FUNCTION_BLOCK SM_LineRegulator EXTENDS StateMachine
VAR_INPUT
	 sSubscription1 : STRING(8);
	 sSubscription2 : STRING(8);
	 sSubscription3 : STRING(8);
END_VAR
VAR_OUTPUT
END_VAR
VAR
	fbTurntable : Turntable;

	aRollerConveyors : ARRAY[1..3] OF RollerConveyor;
	fbRollerConveyorExit : RollerConveyor;
	fbReadyStepWorker : FB_StepWorker;
	fbBusyStepWorker : FB_StepWorker;
	fbInitStepWorker : FB_StepWorker;
	
	messageIndex : UINT;
	stMqttPayload : ST_MqttPayload;
	aSubscriptions : ARRAY[1..3] OF STRING(8);
	uiSubscriptionsCycler : UINT := 1;
END_VAR

SUPER^();
fbTurntable();
aRollerConveyors[1]();
aRollerConveyors[3]();

METHOD PROTECTED   Busy : BOOL
VAR_INPUT
END_VAR
fbBusyStepWorker();
CASE fbBusyStepWorker.uiStep OF

	0:
	
		aRollerConveyors[uiSubscriptionsCycler].On();
		CASE uiSubscriptionsCycler OF
		
			1:
				fbTurntable.RollPlus();
				fbTurntable.Turn();
			
			2:
				fbTurntable.RollPlus();
			
			3:
				fbTurntable.RollMinus();
				fbTurntable.Turn();
		END_CASE
		
		fbBusyStepWorker
			.mAddCondition(itfStepCondition := fbTurntable.fbBackLimit.getSignal)
			.mAddCondition(itfStepCondition := fbTurntable.fbFrontLimit.getSignal)
			.mNextStep(10);
			
	10:
	
		aRollerConveyors[uiSubscriptionsCycler].Off();
		CASE uiSubscriptionsCycler OF
		
			1:
				fbTurntable.StopRolling();			
				fbTurntable.UnTurn();
				fbBusyStepWorker
					.mSetTimer(T#2S)
					.mNextStep(20);
			
			2:
				fbBusyStepWorker.mNextStep(30);
			
			3:
				fbTurntable.StopRolling();
				fbTurntable.UnTurn();
				fbBusyStepWorker
					.mSetTimer(T#2S)
					.mNextStep(20);
		END_CASE
		
	20:
	
		fbTurntable.RollPlus();
		fbRollerConveyorExit.On();
		fbBusyStepWorker
			.mSetTimer(T#2S)
			.mNextStep(30);
	30:	
	
		IF NOT fbTurntable.fbBackLimit.bSignal
			AND NOT fbTurntable.fbFrontLimit.bSignal
		THEN
			fbRollerConveyorExit.Off();
			fbBusyStepWorker
				.mSetTimer(T#1S)
				.mNextStep(40);
		END_IF
		
	40:
	
		fbBusyStepWorker.mNextStep(0);
		Done();
		
	
END_CASE
END_METHOD

METHOD PROTECTED  Error : BOOL
VAR_INPUT
END_VAR
END_METHOD

METHOD PROTECTED  Idle : BOOL
VAR_INPUT
END_VAR
END_METHOD

METHOD PROTECTED  Init : BOOL
VAR_INPUT
END_VAR
fbInitStepWorker();
CASE fbInitStepWorker.uiStep OF

	0: 
	
		IF ADS.fbAdsConnector.isConnected
		THEN
			fbInitStepWorker.mNextStep(10);
		END_IF
		
	10:
	
		IF ADS.fbMqttClient.Subscribe(sSubscription1)
		THEN			
			fbInitStepWorker.mNextStep(20);
		END_IF
		
	20:
	
		IF ADS.fbMqttClient.Subscribe(sSubscription2)
		THEN			
			fbInitStepWorker.mNextStep(30);
		END_IF
		
	30:
		
		IF ADS.fbMqttClient.Subscribe(sSubscription3)
		THEN		
			aSubscriptions[1] := sSubscription1;
			aSubscriptions[2] := sSubscription2;
			aSubscriptions[3] := sSubscription3;
			Start();
		END_IF		
		
END_CASE
END_METHOD

METHOD PROTECTED  Prepare : BOOL
VAR_INPUT
END_VAR
END_METHOD

METHOD PROTECTED  Ready : BOOL
VAR_INPUT
END_VAR
VAR
	
END_VAR
fbReadyStepWorker();

IF uiSubscriptionsCycler = 3
THEN
	uiSubscriptionsCycler := 1;
ELSE
	uiSubscriptionsCycler := uiSubscriptionsCycler + 1;
END_IF

CASE fbReadyStepWorker.uiStep OF

	0: 
		IF NOT fbTurntable.bBackLimit
			AND NOT fbTurntable.bFrontLimit
		THEN
			fbReadyStepWorker.mNextStep(10);
		END_IF
		
	10:
	
		messageIndex := ADS.fbMqttClient.isNewMessage(aSubscriptions[uiSubscriptionsCycler]);
		IF messageIndex > 0
		THEN
			stMqttPayload := Ads.fbMqttClient.getNewMessage(messageIndex);
			fbReadyStepWorker.mNextStep(20);
		END_IF
		
	20:	
		Ads.fbMqttClient.Publish(aSubscriptions[uiSubscriptionsCycler],stMqttPayload);
		fbReadyStepWorker.mNextStep(0);
		Execute();
		
END_CASE
END_METHOD

METHOD PROTECTED  Waiting : BOOL
VAR_INPUT
END_VAR
END_METHOD

END_FUNCTION_BLOCK

(* stored: Version 1.1.0.1, ProductVersion 3.1.4024.2
   POU SM_LineRegulator: Id {ca3d4937-9986-4e8e-b7ee-5deb908a267b}, SpecialFunc None
   Method Busy: Id {5f49f79a-dd7d-411c-abbd-7df000596daa}
   Method Error: Id {239c3776-b310-4e44-8c9a-3b822be85443}
   Method Idle: Id {8991d786-6df6-47cb-9e47-3ad5344b1f79}
   Method Init: Id {61709bba-0e18-44c6-961b-6552433808b6}
   Method Prepare: Id {6b592004-8cf2-4348-b3e7-517e0f77b060}
   Method Ready: Id {f9a8f055-f81d-4c23-82e5-c30d5480dd80}
   Method Waiting: Id {d736384e-810f-4ff5-9820-b539fdf97b0f} *)
